Fanuc TP program (LS listing): INTPULSE.LS

/PROG  INTPULSE
/ATTR
OWNER		= MNEDITOR;
COMMENT		= "IntPulse";
PROG_SIZE	= 0;
CREATE		= DATE 26-01-01  TIME 00:00:00;
MODIFIED	= DATE 26-01-01  TIME 00:00:00;
FILE_NAME	= ;
VERSION		= 0;
LINE_COUNT	= 5;
MEMORY_SIZE	= 0;
PROTECT		= READ_WRITE;
TCD:  STACK_SIZE	= 0,
      TASK_PRIORITY	= 50,
      TIME_SLICE	= 0,
      BUSY_LAMP_OFF	= 0,
      ABORT_REQUEST	= 0,
      PAUSE_REQUEST	= 0;
DEFAULT_GROUP	= 1,*,*,*,*;
CONTROL_CODE	= 00000000 00000000;
/MN
   1:  !RAPID IntProbe.IntPulse ;
   2:  DO[1]=ON ;
   3:  WAIT    .10(sec) ;
   4:  DO[1]=OFF ;
   5:  WAIT    .10(sec) ;
/POS
/END
